// TIA Portal V19 export
TYPE "MotorSAlr"
// stored: Access Published
   STRUCT
      ThermalProtectionA : Bool := FALSE;
      ThermalProtectionB : Bool := FALSE;
      Feedback : Bool := FALSE;
   END_STRUCT;
END_TYPE
